PROGRAM Axis02_Auto
VAR
	Always_ON	:	BOOL	:=TRUE	;//상시 ON 
	Always_OFF	:	BOOL	:=FALSE	;//상시 OFF
END_VAR

// NETWORK 1

END_PROGRAM

(* stored: Version 1.1.0.1, ProductVersion 3.1.4024.15
   POU Axis02_Auto: Id {bb8b8c2e-2fd8-4db4-a00c-53cc54166e35}, SpecialFunc None *)
